TYPE "Positioning_DOL_Machine_Par"
VERSION : 0.1
// Block: Positioning_DOL_Machine_Par
   STRUCT
      PosTolerance : LReal;
      Minus_Limit : LReal;
      Plus_Limit : LReal;
      PreCutOff : LReal;
      PreEndLowSpeed : LReal;
      PreEndMedSpeed : LReal;
      LowSpeed : LReal;
      MedSpeed : LReal;
      HighSpeed : LReal;
      Man_Speed : LReal;
   END_STRUCT;

END_TYPE
